# EPICS autosave request: diffCtrlApp/Db/diff-ctrl.req
## This file specifies which PVs of the corresponding database should be saved.

# Position set points.
# These records do not process at initialization.
$(P)$(R)LeftEdgePos-SP
$(P)$(R)RightEdgePos-SP
$(P)$(R)Center-SP
$(P)$(R)Width-SP

# Tweak step set points
$(P)$(R)RightEdgeStep-SP
$(P)$(R)LeftEdgeStep-SP
$(P)$(R)CenterStep-SP
$(P)$(R)WidthStep-SP
